TYPE DUT_StoredPosition :
STRUCT
	Comment: STRING;
	Position: DUT_COORD_REF;
END_STRUCT
END_TYPE

(* stored: Version 1.1.0.1
   DUT DUT_StoredPosition: Id {66e85fd8-6344-4340-a216-0e3ccb4605b3} *)
